TYPE ST_Service_DigitalOutInWithDependency EXTENDS ST_Service_DigitalOutIn:
STRUCT
	{attribute 'TcHmiSystemEng.Parameter.Name' := 'Dependency state'}
	DependencyOK			: BOOL; 
END_STRUCT
END_TYPE

(* stored: Version 1.1.0.1, ProductVersion 3.1.4026.18
   DUT ST_Service_DigitalOutInWithDependency: Id {b24e9df1-b230-4fa5-a353-d54e008c1808} *)
